(* PLC project Tc2_Utilities.WSTRNCPY Demo, tc3-libraries-kb TwinCAT 3.1 *)
(* stored: creationDateTime 2026-05-12T00:00:00, modificationDateTime 2026-05-12T00:00:00 *)

PROGRAM P_Demo_WSTRNCPY
  VAR
    wsSrc : WSTRING := "HMI text alpha";  (* 工业语义：源 WSTRING *)
    wsDst : WSTRING;  (* 目标 WSTRING *)
    bOk : BOOL;  (* 完整复制 *)
    nSrcLen : UDINT;  (* 源字符数 *)
    nDstLen : UDINT;  (* 目标字符数 *)
    bCopy : BOOL;  (* 在线触发 *)
  END_VAR

// =============================================================================
// 场景：HMI 字符串缓冲动态复制——索引可能越界，比 `:=` 更安全。
// 价值：`Tc2_Standard.WSTRNCPY` ⚠️ 不存在（标准库无对应）——本函数填补 WSTRING 安全复制空缺。
// 验证步骤：
//   1. 引用 Tc2_Utilities
//   2. 编译 + 登录 + 运行
//   3. 在线写触发位 TRUE，monitor 输出变量
// =============================================================================
IF bCopy THEN
    bOk := WSTRNCPY(pDst     := ADR(wsDst),
                    pSrc     := ADR(wsSrc),
                    nDstSize := SIZEOF(wsDst),
                    nSrcLen  => nSrcLen,
                    nDstLen  => nDstLen);
    bCopy := FALSE;
END_IF;
END_PROGRAM
